// Mitsubishi GX Works2 project: 绿灯自动复位   PLC: FX2N/FX2NC

PROGRAM MAIN
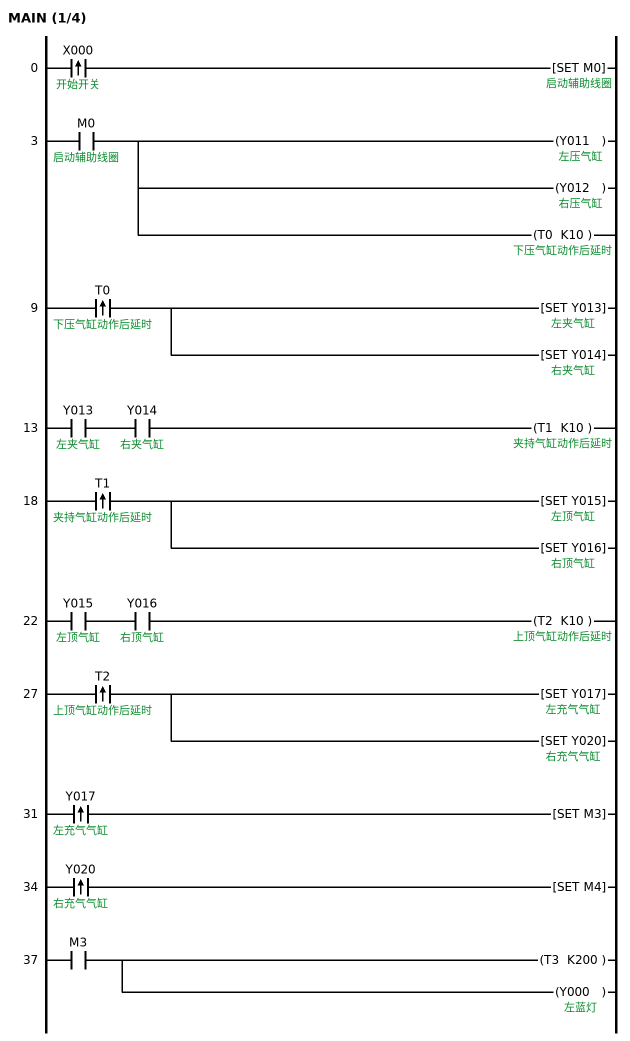
0     LDP     X000  ; 开始开关
      SET     M0  ; 启动辅助线圈
3     LD      M0  ; 启动辅助线圈
      OUT     Y011  ; 左压气缸
      OUT     Y012  ; 右压气缸
      OUT     T0 K10  ; 下压气缸动作后延时
9     LDP     T0  ; 下压气缸动作后延时
      SET     Y013  ; 左夹气缸
      SET     Y014  ; 右夹气缸
13    LD      Y013  ; 左夹气缸
      AND     Y014  ; 右夹气缸
      OUT     T1 K10  ; 夹持气缸动作后延时
18    LDP     T1  ; 夹持气缸动作后延时
      SET     Y015  ; 左顶气缸
      SET     Y016  ; 右顶气缸
22    LD      Y015  ; 左顶气缸
      AND     Y016  ; 右顶气缸
      OUT     T2 K10  ; 上顶气缸动作后延时
27    LDP     T2  ; 上顶气缸动作后延时
      SET     Y017  ; 左充气气缸
      SET     Y020  ; 右充气气缸
31    LDP     Y017  ; 左充气气缸
      SET     M3
34    LDP     Y020  ; 右充气气缸
      SET     M4
37    LD      M3
      OUT     T3 K200
      OUT     Y000  ; 左蓝灯
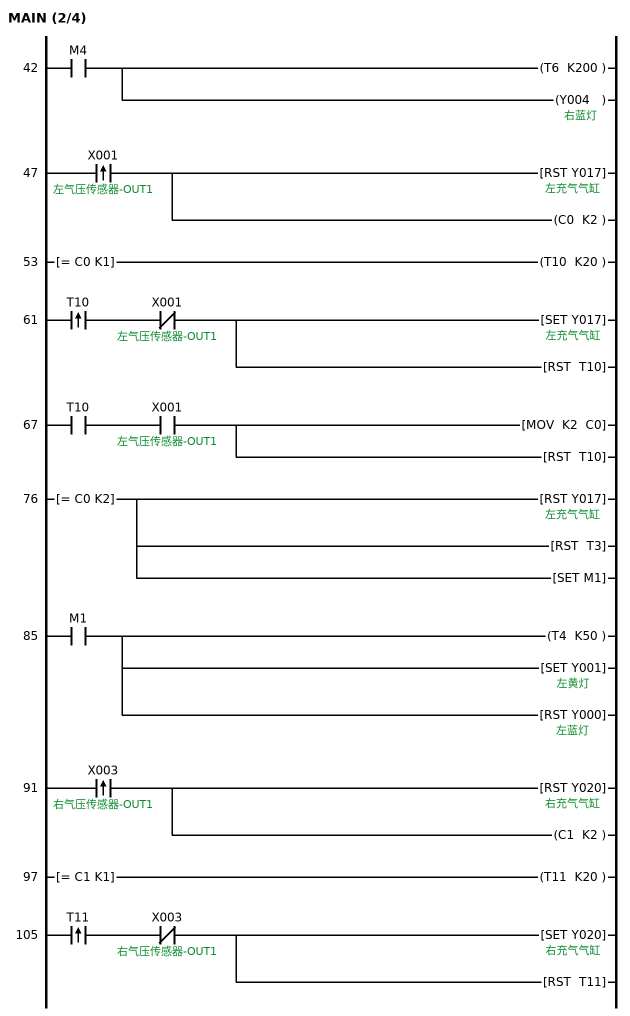
42    LD      M4
      OUT     T6 K200
      OUT     Y004  ; 右蓝灯
47    LDP     X001  ; 左气压传感器-OUT1
      RST     Y017  ; 左充气气缸
      OUT     C0 K2
53    LD=     C0 K1
      OUT     T10 K20
61    LDP     T10
      ANI     X001  ; 左气压传感器-OUT1
      SET     Y017  ; 左充气气缸
      RST     T10
67    LD      T10
      AND     X001  ; 左气压传感器-OUT1
      MOV     K2 C0
      RST     T10
76    LD=     C0 K2
      RST     Y017  ; 左充气气缸
      RST     T3
      SET     M1
85    LD      M1
      OUT     T4 K50
      SET     Y001  ; 左黄灯
      RST     Y000  ; 左蓝灯
91    LDP     X003  ; 右气压传感器-OUT1
      RST     Y020  ; 右充气气缸
      OUT     C1 K2
97    LD=     C1 K1
      OUT     T11 K20
105   LDP     T11
      ANI     X003  ; 右气压传感器-OUT1
      SET     Y020  ; 右充气气缸
      RST     T11
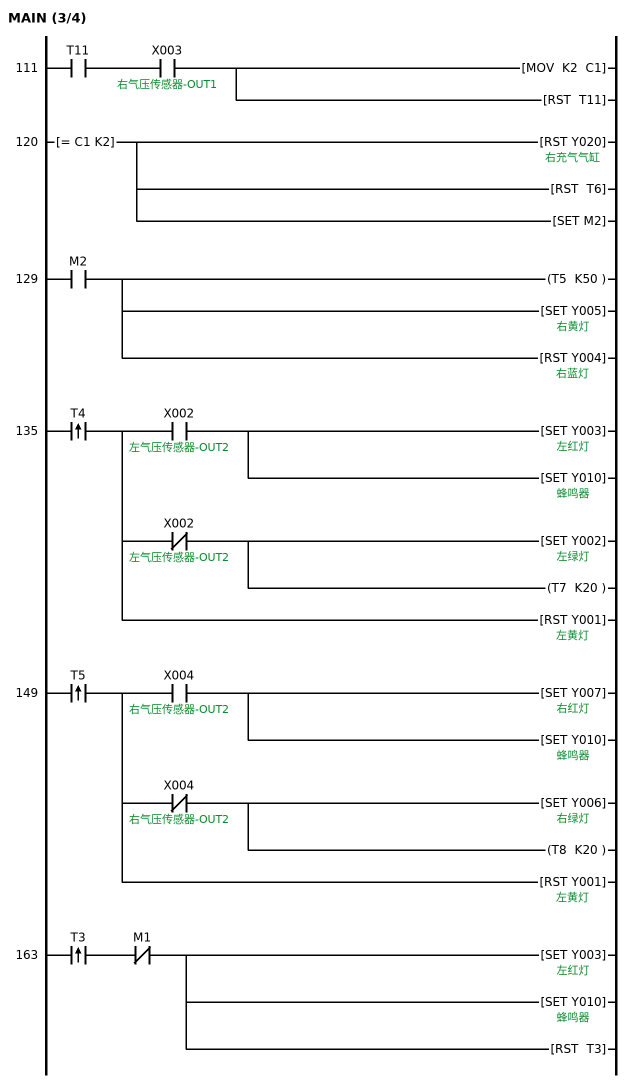
111   LD      T11
      AND     X003  ; 右气压传感器-OUT1
      MOV     K2 C1
      RST     T11
120   LD=     C1 K2
      RST     Y020  ; 右充气气缸
      RST     T6
      SET     M2
129   LD      M2
      OUT     T5 K50
      SET     Y005  ; 右黄灯
      RST     Y004  ; 右蓝灯
135   LDP     T4
      MPS
      AND     X002  ; 左气压传感器-OUT2
      SET     Y003  ; 左红灯
      SET     Y010  ; 蜂鸣器
      MRD
      ANI     X002  ; 左气压传感器-OUT2
      SET     Y002  ; 左绿灯
      OUT     T7 K20
      MPP
      RST     Y001  ; 左黄灯
149   LDP     T5
      MPS
      AND     X004  ; 右气压传感器-OUT2
      SET     Y007  ; 右红灯
      SET     Y010  ; 蜂鸣器
      MRD
      ANI     X004  ; 右气压传感器-OUT2
      SET     Y006  ; 右绿灯
      OUT     T8 K20
      MPP
      RST     Y001  ; 左黄灯
163   LDP     T3
      ANI     M1
      SET     Y003  ; 左红灯
      SET     Y010  ; 蜂鸣器
      RST     T3
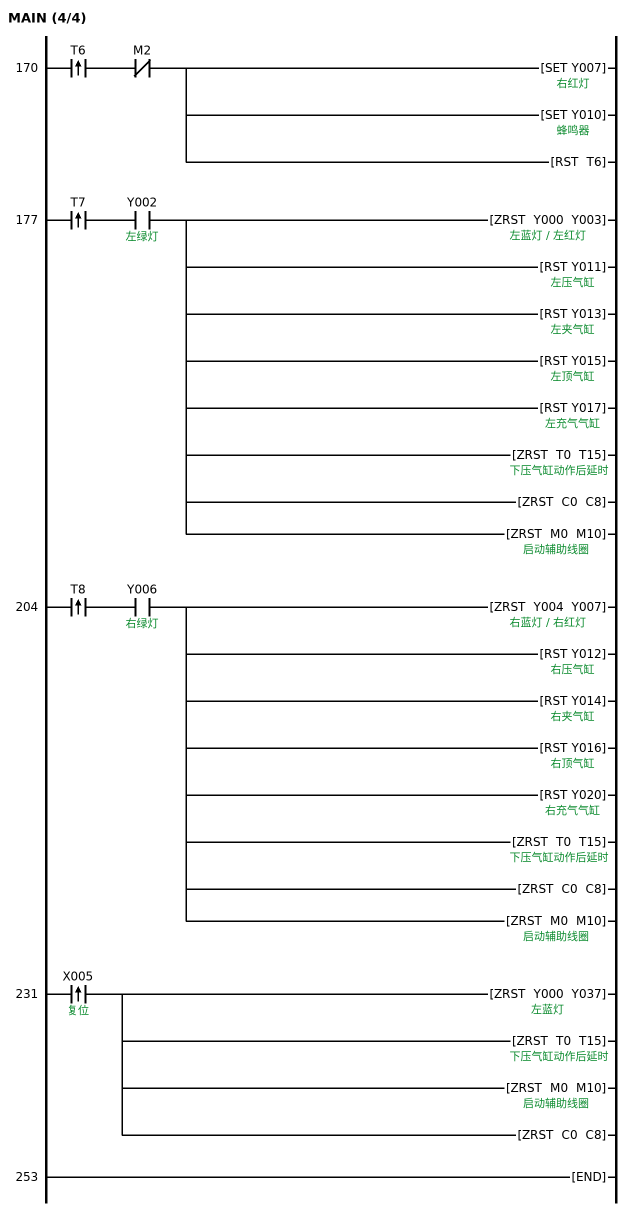
170   LDP     T6
      ANI     M2
      SET     Y007  ; 右红灯
      SET     Y010  ; 蜂鸣器
      RST     T6
177   LDP     T7
      AND     Y002  ; 左绿灯
      ZRST    Y000 Y003
      RST     Y011  ; 左压气缸
      RST     Y013  ; 左夹气缸
      RST     Y015  ; 左顶气缸
      RST     Y017  ; 左充气气缸
      ZRST    T0 T15
      ZRST    C0 C8
      ZRST    M0 M10
204   LDP     T8
      AND     Y006  ; 右绿灯
      ZRST    Y004 Y007
      RST     Y012  ; 右压气缸
      RST     Y014  ; 右夹气缸
      RST     Y016  ; 右顶气缸
      RST     Y020  ; 右充气气缸
      ZRST    T0 T15
      ZRST    C0 C8
      ZRST    M0 M10
231   LDP     X005  ; 复位
      ZRST    Y000 Y037
      ZRST    T0 T15
      ZRST    M0 M10
      ZRST    C0 C8
253   END
END_PROGRAM
